FUNCTION_BLOCK tf_3 (* Basic FB with empty ECC *)
  (* Standard: 61499-2 *)
  (* Version 1.0, 2021-03-12, Lenovo *)
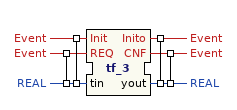
  EVENT_INPUT
    Init WITH tin;
    REQ WITH tin;
  END_EVENT
  EVENT_OUTPUT
    Inito WITH yout;
    CNF WITH yout;
  END_EVENT
  VAR_INPUT
    tin : REAL;
  END_VAR
  VAR_OUTPUT
    yout : REAL;
  END_VAR
  VAR
    x : REAL; (* Internal Variable *)
    n : REAL; (* Internal Variable *)
  END_VAR
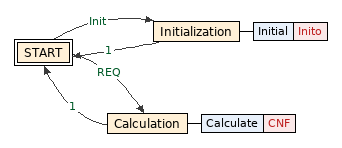
  EC_STATES
    START; (* Initial State *)
    Initialization : Initial -> Inito;
    Calculation : Calculate -> CNF;
  END_STATES
  EC_TRANSITIONS
    START TO Initialization := Init;
    Initialization TO START := 1;
    START TO Calculation := REQ;
    Calculation TO START := 1;
  END_TRANSITIONS
  ALGORITHM Initial IN ST: (* New Algorithm *)

  END_ALGORITHM
  ALGORITHM Calculate IN ST: (* New Algorithm *)
x:=-tin;
n:=EXP(x);
yout:=(1)*n;
  END_ALGORITHM
END_FUNCTION_BLOCK
